# B&R Automation Studio project Lecture_06_homework
Automation Studio 4.8.2.72

## Configuration Config1

### Hardware
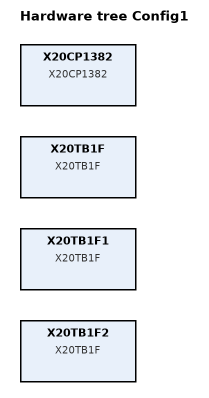
```
X20CP1382 : X20CP1382 v1.10.0.0  [X1 -> X1.SL; X2 -> X2.SL; X3 -> X3.SL]
  Module X1 (Type=X1, Virtual=true, Version=1.10.0.0)
    Connection (Connector=SS1, TargetModule=X20TB1F, TargetConnector=SS)
    Connection (Connector=SL, TargetModule=X20CP1382, TargetConnector=X1)
  Module X2 (Type=X2, Virtual=true, Version=1.10.0.0)
    Connection (Connector=SS1, TargetModule=X20TB1F1, TargetConnector=SS)
    Connection (Connector=SL, TargetModule=X20CP1382, TargetConnector=X2)
  Module X3 (Type=X3, Virtual=true, Version=1.10.0.0)
    Connection (Connector=SS1, TargetModule=X20TB1F2, TargetConnector=SS)
    Connection (Connector=SL, TargetModule=X20CP1382, TargetConnector=X3)
  Connector IF2:
    ActivateDevice = 1
  Simulation = 1
X20TB1F : X20TB1F v1.0.0.0
X20TB1F1 : X20TB1F v1.0.0.0
X20TB1F2 : X20TB1F v1.0.0.0
```

## Logical view

### Program Logical/Program

#### Main.st
```iecst
PROGRAM _INIT
	// Assignment 2 - Bit shifting
	VAR
		aBit_shifting : ARRAY[0..15] OF BOOL;
	END_VAR
	aBit_shifting[15] := TRUE;

END_PROGRAM

PROGRAM _CYCLIC
	(* Insert code here *)
	// Assignment 1 - Alternating light
	A := A + 1;

	// Assignment 2 - Bit shifting

END_PROGRAM

PROGRAM _EXIT
	(* Insert code here *)

END_PROGRAM
```
